// Block: AreaGen_Messages

DATA_BLOCK AreaGen_Messages
VERSION : 0.1
   NON_RETAIN
   VAR
      A : Struct
         Msg : Array[1..304] of Bool;
         Hmi : Array[1..19] of Word;
         Ack : Array[1..19] of Word;
      END_STRUCT;
      W : Struct
         Msg : Array[1..256] of Bool;
         Hmi : Array[1..16] of Word;
         Ack : Array[1..16] of Word;
      END_STRUCT;
      Area01_A_Counter : Int;
      Area01_W_Counter : Int;
      Area02_A_Counter : Int;
      Area02_W_Counter : Int;
      Area03_A_Counter : Int;
      Area03_W_Counter : Int;
   END_VAR

BEGIN
   // No initialization required
END_DATA_BLOCK
